  def rq_gripper_led_force_purple(gripper_socket="1"):
      rq_set_var(LBP,1, gripper_socket)
      rq_set_var(LRD,1, gripper_socket)
      rq_set_var(LBL,1, gripper_socket)
      rq_set_var(LGN,0, gripper_socket)
  end

  ############################################
  # mm/inches functions
  ############################################
  gripper_closed_norm = [100, 100, 100, 100]
  gripper_open_norm = [0, 0, 0, 0]
  gripper_closed_mm = [0, 0, 0, 0]
  gripper_open_mm = [50, 50, 50, 50]

  def rq_current_pos_mm(gripper_socket=1):
      pos_gripper = rq_current_pos(gripper_socket)
      pos_mm = gripper_to_mm(pos_gripper, gripper_socket)
      return round_value_2_dec(pos_mm)
  end

  def rq_current_pos_inches(gripper_socket=1):
      pos_gripper = rq_current_pos(gripper_socket)
      pos_mm = gripper_to_mm(pos_gripper, gripper_socket)
      pos_in = pos_mm / 25.4
      return round_value_2_dec(pos_in)
  end

  def rq_move_mm(pos_mm, gripper_socket=1):
      pos_gripper = mm_to_gripper(pos_mm, gripper_socket)
      rq_move(pos_gripper, gripper_socket)
  end

  def rq_move_and_wait_mm(pos_mm, gripper_socket=1):
      pos_gripper = mm_to_gripper(pos_mm, gripper_socket)
      rq_move_and_wait(pos_gripper, gripper_socket)
  end

  def rq_move_inches(pos_in, gripper_socket=1):
      pos_mm = pos_in * 25.4
      rq_move_mm(pos_mm, gripper_socket)
  end

  def rq_move_and_wait_inches(pos_in, gripper_socket=1):
      pos_mm = pos_in * 25.4
      rq_move_and_wait_mm(pos_mm, gripper_socket)
  end

  def get_closed_norm(gripper_socket):
      return gripper_closed_norm[gripper_socket - 1]
  end

  def get_open_norm(gripper_socket):
      return gripper_open_norm[gripper_socket - 1]
  end

  def get_closed_mm(gripper_socket):
      return gripper_closed_mm[gripper_socket - 1]
  end

  def get_open_mm(gripper_socket):
      return gripper_open_mm[gripper_socket - 1]
  end

  def set_closed_norm(closed_norm, gripper_socket):
      gripper_closed_norm[gripper_socket - 1] = closed_norm
  end

  def set_open_norm(open_norm, gripper_socket):
      gripper_open_norm[gripper_socket - 1] = open_norm
  end

  def set_closed_mm(closed_mm, gripper_socket):
      gripper_closed_mm[gripper_socket - 1] = closed_mm
  end

  def set_open_mm(open_mm, gripper_socket):
      gripper_open_mm[gripper_socket - 1] = open_mm
  end

  def gripper_to_mm(value_gripper, gripper_socket):
      closed_norm = get_closed_norm(gripper_socket)
      open_norm = get_open_norm(gripper_socket)
      closed_mm = get_closed_mm(gripper_socket)
      open_mm = get_open_mm(gripper_socket)

      value_norm = (value_gripper / 255) * 100

      slope = (closed_mm - open_mm) / (closed_norm - open_norm)
      value_mm = slope * (value_norm - closed_norm) + closed_mm

      if (value_mm > open_mm):
          value_mm_limited = open_mm
      elif (value_mm < closed_mm):
          value_mm_limited = closed_mm
      else:
          value_mm_limited = value_mm
      end

      return value_mm_limited
  end

  def mm_to_gripper(value_mm, gripper_socket):
      closed_norm = get_closed_norm(gripper_socket)
      open_norm = get_open_norm(gripper_socket)
      closed_mm = get_closed_mm(gripper_socket)
      open_mm = get_open_mm(gripper_socket)

      slope = (closed_norm - open_norm) / (closed_mm - open_mm)
      value_norm = (value_mm - closed_mm) * slope + closed_norm

      value_gripper = value_norm * 255 / 100

      if (value_gripper > 255):
          value_gripper_limited = 255
      elif (value_gripper < 0):
          value_gripper_limited = 0
      else:
          value_gripper_limited = round_value(value_gripper)
      end

      return value_gripper_limited
  end

  def round_value(value):
      value_mod = value % 1

      if(value_mod < 0.5):
          return floor(value)
      else:
          return ceil(value)
      end
  end

  def round_value_2_dec(value):
      value_x_100 = value * 100
      value_x_100_rounded = round_value(value_x_100)
      return value_x_100_rounded / 100
  end

  def clear_socket_buffer(gripper_socket="1", read_timeout = 0.1):
    byte_in_buffer = socket_read_byte_list(1, gripper_socket, read_timeout)

    while(byte_in_buffer[0] >= 1):
        byte_in_buffer = socket_read_byte_list(1, gripper_socket, read_timeout)
    end
  end

  def rq_set_gripper_socket_acquire_option(enabled=False):
      gripper_socket_acquire_option = enabled

      if(not enabled):
          gripper_1_socket_acquired = False
          gripper_2_socket_acquired = False
          gripper_3_socket_acquired = False
          gripper_4_socket_acquired = False
      end
  end

  def rq_acquire_gripper_socket(gripper_socket="1"):
      if(gripper_socket_acquire_option):
          rq_wait_gripper_socket_released(gripper_socket)
          enter_critical
              rq_set_gripper_socket_acquired(gripper_socket, True)
          exit_critical

          clear_socket_buffer(gripper_socket, 0.002)

          sync()
      end
  end

  def rq_release_gripper_socket(gripper_socket="1"):
      if(gripper_socket_acquire_option):
          rq_set_gripper_socket_acquired(gripper_socket, False)

          sync()
      end
  end

  def rq_set_gripper_socket_acquired(gripper_socket="1", acquired=False):
      if(gripper_socket == "1"):
          gripper_1_socket_acquired = acquired
      elif(gripper_socket == "2"):
          gripper_2_socket_acquired = acquired
      elif(gripper_socket == "3"):
          gripper_3_socket_acquired = acquired
      elif(gripper_socket == "4"):
          gripper_4_socket_acquired = acquired
      end
  end

  def rq_get_gripper_socket_acquired(gripper_socket="1"):
      if(gripper_socket == "1"):
          return gripper_1_socket_acquired
      elif(gripper_socket == "2"):
          return gripper_2_socket_acquired
      elif(gripper_socket == "3"):
          return gripper_3_socket_acquired
      elif(gripper_socket == "4"):
          return gripper_4_socket_acquired
      end

      sync()
  end

  def rq_wait_gripper_socket_released(gripper_socket="1"):
      while(rq_get_gripper_socket_acquired(gripper_socket)):
          sync()
      end

      sync()
  end

  def rq_gripper_id_to_ascii(gripper_id):
      if(gripper_id == "1"):
          return 57
      elif(gripper_id == "2"):
          return 50
      elif(gripper_id == "3"):
          return 51
      elif(gripper_id == "4"):
          return 52
      end
  end

  def scale(value, rawRange, scaledRange):
      def computeSlope(inputRange, outputRange):
          outputRangeDelta = outputRange[1] - outputRange[0]
          inputRangeDelta = inputRange[1] - inputRange[0]

          if (inputRangeDelta == 0):
              return 0
          else:
              return outputRangeDelta / inputRangeDelta
          end
      end

      def computeIntercept(slope, inputRange, outputRange):
          return outputRange[0] - (slope * inputRange[0])
      end

      def clipScaledValue(outputScaledValue, outputRange):
          if (outputRange[0] < outputRange[1]):
              return clipWhenLowerLimitIsLessThanHigher(outputScaledValue, outputRange)
          else:
              return clipWhenLowerLimitIsGreaterThanHigherLimit(outputScaledValue, outputRange)
          end
      end

      def clipWhenLowerLimitIsGreaterThanHigherLimit(outputScaledValue, outputRange):
          if (outputScaledValue < outputRange[1]):
              return outputRange[1]
          elif (outputScaledValue > outputRange[0]):
              return outputRange[0]
          else:
              return outputScaledValue
          end
      end

      def clipWhenLowerLimitIsLessThanHigher(outputScaledValue, outputRange):
          if (outputScaledValue < outputRange[0]):
              return outputRange[0]
          elif (outputScaledValue > outputRange[1]):
              return outputRange[1]
          else:
              return outputScaledValue
          end
      end

      slope = computeSlope(rawRange, scaledRange)
      intercept = computeIntercept(slope, rawRange, scaledRange)
      scaledValue = slope * value + intercept
      return clipScaledValue(scaledValue, scaledRange)
  end

  def limit(value, range):
      return scale(value, range, range)
  end


  rq_obj_detect = 0
  set_tool_voltage(24)
  set_tool_communication(True, 115200, 0, 1, 1.5, 3.5)
  rq_wait_for_gripper_connected()
  rq_init_comm_if_connected(9, "1")
  rq_init_comm_if_connected(2, "2")
  rq_init_comm_if_connected(3, "3")
  rq_init_comm_if_connected(4, "4")
  rq_print_connected_grippers()
  connectivity_checked = [-1,-1,-1,-1]
  status_checked = [-1,-1,-1,-1]
  current_speed = [-1,-1,-1,-1]
  current_force = [-1,-1,-1,-1]
  set_closed_norm(90.19607843137254, 1)
  set_open_norm(1.1764705882352942, 1)
  set_closed_mm(0.0, 1)
  set_open_mm(143.0, 1)
  set_closed_norm(100.0, 2)
  set_open_norm(0.0, 2)
  set_closed_mm(0.0, 2)
  set_open_mm(50.0, 2)
  set_closed_norm(100.0, 3)
  set_open_norm(0.0, 3)
  set_closed_mm(0.0, 3)
  set_open_mm(50.0, 3)
  set_closed_norm(100.0, 4)
  set_open_norm(0.0, 4)
  set_closed_mm(0.0, 4)
  set_open_mm(50.0, 4)
  # end: URCap Installation Node
  $ 1 "Robot Program"
  $ 2 "Script: artmDemofast_all.script"
      g_ftRaw = [0, 0, 0, 0, 0, 0, 0]
      g_transFlangeFts = pose_inv(p[0, 0, 0, 0, 0, 0])
      g_extFTRcv_stopReq = False
      g_filterOn = True

      set_payload(get_target_payload(), get_target_payload_cog())

      def filterData(a, b, currentPose, previousPose):
          counter = 0
          pose = currentPose
          if g_filterOn:
              while(counter < 6):
                  pose[counter] = (a * currentPose[counter] + b * previousPose[counter]) /(a + b)
                  counter = counter + 1
              end
          end
          return pose
      end

      thread extFTReceiverThread():
          prevData = p[0,0,0,0,0,0]
          while g_extFTRcv_stopReq == False:
              Error = 0
              ftRawData = get_tcp_force()
              ftRawData = filterData(0.002, 0.05, ftRawData, prevData)
              prevData = ftRawData

              flangePose = pose_inv(get_actual_tool_flange_pose())
              flangePose = p[0.0, 0.0, 0.0, flangePose[3], flangePose[4], flangePose[5]]

              ftDataForce = p[ftRawData[0], ftRawData[1], ftRawData[2], 0.0, 0.0, 0.0]
              ftDataForce = pose_trans(g_transFlangeFts,  pose_trans(flangePose, ftDataForce))

              ftDataTorque = p[ftRawData[3], ftRawData[4], ftRawData[5], 0.0, 0.0, 0.0]
              ftDataTorque = pose_trans(g_transFlangeFts, pose_trans(flangePose, ftDataTorque))
              enter_critical
              g_ftRaw = [Error, ftDataForce[0], ftDataForce[1], ftDataForce[2], ftDataTorque[0], ftDataTorque[1], ftDataTorque[2]]
              exit_critical
              sync()
          end
      end

      fts_rcv_thread = run extFTReceiverThread()

      # make sure we receive FT data
      while g_extFTRcv_stopReq == False:
          enter_critical
          tmpForceZ = g_ftRaw[3]
          exit_critical
          if tmpForceZ != 0:
             textmsg("ok, got some real force data")
             break
          end
          sync()
      end

      def killExtFTReceiverThread():
          kill fts_rcv_thread
      end
      g_ftRawBias_0 = 0
      g_ftRawBias_1 = 0
      g_ftRawBias_2 = 0
      g_ftRawBias_3 = 0
      g_ftRawBias_4 = 0
      g_ftRawBias_5 = 0
      def setExtFTBias():
          textmsg("Sleeping 0.1s to set Bias")
          sleep(0.1)
          # TODO: we need a more robust bias
          enter_critical
          local tmp = g_ftRaw
          exit_critical
          # use strongly smoothed data
          g_ftRawBias_0 = tmp[1]
          g_ftRawBias_1 = tmp[2]
          g_ftRawBias_2 = tmp[3]
          g_ftRawBias_3 = tmp[4]
          g_ftRawBias_4 = tmp[5]
          g_ftRawBias_5 = tmp[6]
          return tmp
      end

      def servojToTarget_132(target, a, v, t):
          local jp = get_target_joint_positions()
          i = 50
          if (t < 0.008):
              t = 0.008
          end
          while ((norm(jp[0] - target[0]) > 0.0006) or
                 (norm(jp[1] - target[1]) > 0.0006) or
                 (norm(jp[2] - target[2]) > 0.0006) or
                 (norm(jp[3] - target[3]) > 0.0006) or
                 (norm(jp[4] - target[4]) > 0.0006) or
                 (norm(jp[5] - target[5]) > 0.0006)) and (i > 0):
              if (evalGlobalConstraints_134()):
                  return True
              end
              servoj(target, a, v, t)
              jp = get_target_joint_positions()
              i = i - 1
          end
          if (i == 0):
              textmsg("servojToTarget: target not reached")
              halt
          end
      end

      def servojToTarget_123(target, a, v, t):
          local jp = get_target_joint_positions()
          i = 50
          if (t < 0.008):
              t = 0.008
          end
          while ((norm(jp[0] - target[0]) > 0.0006) or
                 (norm(jp[1] - target[1]) > 0.0006) or
                 (norm(jp[2] - target[2]) > 0.0006) or
                 (norm(jp[3] - target[3]) > 0.0006) or
                 (norm(jp[4] - target[4]) > 0.0006) or
                 (norm(jp[5] - target[5]) > 0.0006)) and (i > 0):
              if (evalGlobalConstraints_125()):
                  return True
              end
              servoj(target, a, v, t)
              jp = get_target_joint_positions()
              i = i - 1
          end
          if (i == 0):
              textmsg("servojToTarget: target not reached")
              halt
          end
      end


      socket_close("socket_gripper")
      socket_gripper_ok = socket_open("127.0.0.1", 63352, "socket_gripper")
      if socket_gripper_ok == False:
          # exit program/function
          halt
      end
      rps_rq_actual_pos = 1

      # Returns True if list_of_bytes is [3, 'a', 'c', 'k']
      def rps_is_ack(list_of_bytes):

          # list length is not 3
          if (list_of_bytes[0] != 3):
              return False
          end

          # first byte not is 'a'?
          if (list_of_bytes[1] != 97):
              return False
          end

          # first byte not is 'c'?
          if (list_of_bytes[2] != 99):
              return False
          end

          # first byte not is 'k'?
          if (list_of_bytes[3] != 107):
              return False
          end

          return True
      end

      def rps_rq_set_var(var_name, var_value):

          sync()
          socket_set_var(var_name , var_value, "socket_gripper")
          sync()
          ack = socket_read_byte_list(3, "socket_gripper")
          sync()

          while(not rps_is_ack(ack)):

              socket_set_var(var_name , var_value,"socket_gripper")
              sync()
              ack = socket_read_byte_list(3, "socket_gripper")
              sync()
          end
      end

      def rps_rq_get_var(var_name):

          if (var_name == "FLT"):
              socket_send_string("GET FLT","socket_gripper")
          elif (var_name == "OBJ"):
              socket_send_string("GET OBJ","socket_gripper")
          elif (var_name == "STA"):
              socket_send_string("GET STA","socket_gripper")
          elif (var_name == "PRE"):
              socket_send_string("GET PRE","socket_gripper")
          elif (var_name == "GTO"):
              socket_send_string("GET GTO", "socket_gripper")
          else:
              # nothing
          end

          sync()
          var_value = socket_read_byte_list(3, "socket_gripper")
          sync()

          return var_value
      end

      def rps_rq_set_GTO_sync(value):
          rps_rq_set_var("GTO",1)

          while (not rps_rq_is_GTO(value, rps_rq_get_var("GTO"))):
              sync()
          end
      end

      def rps_rq_is_GTO(value, bytes):
          asciiZero = 48

          if (bytes[0] == 1):
              if (bytes[1] == asciiZero + value):
                  return True
              end
          end

          return False
      end

      def regulateVacuum(maxLevel, timeout, minLevel):
          gripperPos = 0
          detectTimeout = 30
          advMode = False

          if (maxLevel == 0):
              gripperPos = 75
          elif (maxLevel == 1 and advMode):
              detectTimeout = 255
          end
          rps_rq_set_var("FOR", 100 - minLevel)
          rps_rq_set_var("POS", 100 - gripperPos)
          rps_rq_set_var("SPE", detectTimeout)

          rps_rq_set_var("MOD", 0)

          rps_rq_set_GTO_sync(1)
      end

      def rps_rq_get_position():

          rps_rq_actual_pos = 1
          if (rps_rq_is_object_detected()):
              rps_rq_actual_pos = 0
          end
          return rps_rq_actual_pos
      end

      # Returns True if list_of_byte is [1, '1'] or [1, '2']
      # Used to test OBJ = 0x1 or OBJ = 0x2
      def rps_is_OBJ_object_detected (list_of_bytes):
          # list length is not 1
          if (list_of_bytes[0] != 1):
              return False
          end

          # byte is '2'?
          if (list_of_bytes[1] == 50):
              return True
          end

          # byte is '1'?
          if (list_of_bytes[1] == 49):
              return True
          end

          return False
      end

      def rps_rq_wait_for_object_not_detected():
          while (rps_rq_is_object_detected()):
              sleep(0.01)
              sync()
          end
      end

      def rps_rq_wait_for_object_detected():
          while (not rps_rq_is_object_detected()):
              if (rps_rq_is_timeout()):
                  return False
              end
          end
          return True
      end

      def rps_rq_is_object_detected():
          gOBJ = rps_rq_get_var("OBJ")

          if(rps_is_OBJ_object_detected(gOBJ)):
              rps_rq_actual_pos = 0
              return True
          else:
              rps_rq_actual_pos = 1
              return False
          end
      end

      def rps_rq_is_timeout():
        return rps_rq_is_FLT(6, rps_rq_get_var("FLT"))
      end

      def rps_rq_is_FLT(fault_number, list_of_bytes):
          zero_ascii = 48
          if (list_of_bytes[0] != 2):
             return False
          end

          if (list_of_bytes[1] != zero_ascii):
              return False
          end

          if (list_of_bytes[2] != zero_ascii + fault_number):
              return False
          end

          return True
      end


      def rps_is_STA_gripper_activated(list_of_bytes):
          # list length is not 1
          if (list_of_bytes[0] != 1):
              return False
          end

          # byte is '3'?
          if (list_of_bytes[1] == 51):
              return True
          end
          return False
      end

      def rps_rq_is_gripper_activated():
          gSTA = rps_rq_get_var("STA")
          return rps_is_STA_gripper_activated(gSTA)
      end

      def rps_rq_activate():
          if (rps_rq_is_gripper_activated()):
              return True
          end
          popup("Gripper is not initialized. Initialize and continue?", title="Gripper Warning", warning=True, error=False, blocking=True)
          # reset
          rps_rq_mov_complete = 0
          rps_rq_obj_detect = 0
          rps_rq_actual_pos = 1
          rps_rq_set_var("ACT", 0)
          rps_rq_set_var("ATR", 0)
          sync()
          # activate
          rps_rq_set_var("ACT", 1)
          while (not rps_rq_is_gripper_activated()):
              # wait for activation completed
              sync()
          end
      end
      rps_rq_activate()
      rps_rq_get_position()

      def gripperMove(pos, speed, force):
          regulateVacuum(pos, speed, 65)

          if (pos == 1):
              global g_errorMoveGripper = False
          elif (pos == 0):
              global g_errorMoveGripper = not rps_rq_wait_for_object_detected()
          end

          return True
      end
      def gripperMoveV2(pos, speed):
          return gripperMove(pos, speed, 65)
      end


      global g_detector_pre_bytes = 4
      global g_detector_max_poses = 16    # determines the data size
      global g_detector_pose_bytes = 8
      global g_time_out_flag_vision = 0
      global g_detector_result = p[0,0,0,0,0,0]

      def RPS_socketTestVision(socket_ok, message):
          if socket_ok == 0:
              # exit program/function
              textmsg("The connection to the camera failed. The programm will be stopped.")
              #halt
              return 0
          else:
              textmsg(message)
              return 1
          end
      end

      def RPS_closeSocketsVision(socket_visor_ok, socket_visor_name):
          if socket_visor_ok == 1:
              socket_close(socket_visor_name)
              socket_visor_ok = 0
          end
          return socket_visor_ok
      end
      global g_detector_max_jobs_cognex = 99

      def sendToCognex(message1, message2, socket):
      	send_ok = socket_send_string(message1, socket)
      	send_ok = send_ok and socket_send_string(message2, socket)
      	send_ok = send_ok and socket_send_byte(13, socket)
      	send_ok = send_ok and socket_send_byte(10, socket)
      	return send_ok
      end

      def sendNumberToCognex(message1, number1, socket):
      	send_ok = socket_send_string(message1, socket)
      	send_ok = send_ok and socket_send_byte(48 + floor(number1 / 10), socket)
      	send_ok = send_ok and socket_send_byte(48 + (number1 % 10), socket)
      	send_ok = send_ok and socket_send_byte(13, socket)
      	send_ok = send_ok and socket_send_byte(10, socket)
      	return send_ok
      end

      def RPS_loginCognex(user, password, socket):
      	strWelcome = socket_read_line(socket)

      	strUser = socket_read_string(socket)
      	if sendToCognex(user, "", socket):
      		strPassword = socket_read_string(socket)
      		if sendToCognex(password, "", socket):
      			strUserLoggedIn = socket_read_line(socket)
      			if strUserLoggedIn == "User Logged In":
      				textmsg( strWelcome )
      				return 1
      			else:
      				textmsg("Login failed, user or password is invalid.")
      				return 0
      			end
      		end
      	end
      	textmsg("Login failed, couldn't send the login messages.")
      	return 0
      end

      def getAsciiToNumber_13_10(socket):
      #reads from a socket ASCII characters and generates Integers from it.
      #The numbers must end with the ASCII-bytes '13', '10'
      	i = 0
      	number = 0
      	sign = 1
      	while True:
      		ascii = socket_read_byte_list(1, socket)
      		if ascii[1] > 47 and ascii[1] < 58:
      			number = number * 10
      			number = number + (ascii[1] - 48)
      		elif ascii[1] == 240 and i == 0:
      			sign = -1
      		elif ascii[1] == 13:
      			ascii = socket_read_byte_list(1, socket)
      			if ascii[1] == 10:
      				return [1, number*sign]
      			else:
      				return [0, 0]
      			end
      		else:
      			return [0, 0]
      		end
      		i = i + 1
      	end
      	return [0, 0]
      end

      def setTriggerCognex(socket):
      	#holding time for the response of the trigger is 2s
      	if sendToCognex("SW8", "", socket):
      		strResponseSetTrg = socket_read_line(socket)
      		if strResponseSetTrg  == "1":
      			return 1
      		else:
      			textmsg("Trigger failed. The camera sent the following error code: ")
      			if strResponseSetTrg == "-2":
      				textmsg("-2: The command could not be executed.")
      				textmsg("Make sure that the trigger of the job is set to 'manual'.")
      			elif strResponseSetTrg == "-6":
      				textmsg("-6: User does not have 'Full Access' to execute the command.")
      			else:
      				textmsg(strResponseSetTrg)
      				textmsg("To decipher the code, please look into the cognex manual at Set Online in Basic Native Mode Communication")
      			end
      			return 0
      		end
      	else:
      		textmsg("Trigger failed, couldn't send the message.")
      		return 0
      	end
      end

      def setOnlineCognex(mode, socket):
      	if sendToCognex("SO", mode, socket):
      		strResponseSetOnl = socket_read_line(socket)
      		if strResponseSetOnl  == "1":
      			return 1
      		else:
      			textmsg("The camera online mode can't be set to: ", mode)
      			textmsg("Set Online failed. The camera sent the following error code: ")
      			if strResponseSetOnl == "-2":
      				textmsg("-2: The command could not be executed.")
      			elif strResponseSetOnl == "-5":
      				textmsg("-5: The communications flag was succesful but the sensor did not go Online because the sensor is set Offline manually.")
      				textmsg("The manual setting could be done through the In-Sight Explorer user interface or by a Discrete I/O signal.")
      			elif strResponseSetOnl == "-6":
      				textmsg("-6: User does not have 'Full Access' to execute the command.")
      			else:
      				textmsg(strResponseSetOnl)
      				textmsg("To decipher the code, please look into the cognex manual at Set Online in Basic Native Mode Communication")
      			end
      			return 0
      		end
      	else:
      		textmsg("Set Online failed, couldn't send the message.")
      		return 0
      	end
      end

      def getJobCognex(socket):
      	if sendToCognex("GJ", "", socket):
      		strResponseGetJob = socket_read_line(socket)
      		if strResponseGetJob  == "1":
      			numResponseGetJob = getAsciiToNumber_13_10(socket)
      			if numResponseGetJob[0] == 1: #actual Jobnumber == numResponseGetJob[1]
      				return numResponseGetJob
      			else:
      				textmsg("Get job failed, couldn't read the answer from the camera.")
      			end
      		else:
      			textmsg("Get job failed. The camera sent the following error code: ", strResponseGetJob)
      			textmsg("To decipher the code, please look into the cognex manual at Get Job in Basic Native Mode Communication")
      			return [0, 0]
      		end
      	else:
      		textmsg("Get job failed, couldn't send the message.")
      		return [0, 0]
      	end
      end

      def setJobCognex(jobnumber, socket):
      	if jobnumber > g_detector_max_jobs_cognex:
      		textmsg("The job index is higher than the supported number of jobs, which is ", g_detector_max_jobs_cognex)
      		return 0
      	end
      	setOnlineCognex("0", socket)
      	if sendNumberToCognex("SJ", jobnumber, socket): #consider timeout, if more than 2s load time
      		strSJ = ""
      		i = 0
      		while strSJ == "":
      			strSJ = socket_read_line(socket)
      			i = i + 1
      			if i == 3 and strSJ == "":
      				strSJ = "0"
      				textmsg("Job change failed. The camera didn't answer anymore.")
      			end
      		end
      		if strSJ == "1":
      			setOnlineCognex("1", socket)
      			return 1
      		else:
      			textmsg("Job change failed. Please check the job number.")
      			return 0
      		end
      	else:
      		textmsg("Job change failed, couldn't send the message.")
      		return 0
      	end
      end

      def invalidateCameraData():
      	sync()
      	# 4+g_detector_max_poses*8 entries
      	return [ 0,0,0,0, 0,0,0,0,0,0,0,0,  0,0,0,0,0,0,0,0,  0,0,0,0,0,0,0,0,  0,0,0,0,0,0,0,0,  0,0,0,0,0,0,0,0,  0,0,0,0,0,0,0,0,  0,0,0,0,0,0,0,0,  0,0,0,0,0,0,0,0,  0,0,0,0,0,0,0,0,  0,0,0,0,0,0,0,0,  0,0,0,0,0,0,0,0,  0,0,0,0,0,0,0,0,  0,0,0,0,0,0,0,0,  0,0,0,0,0,0,0,0,  0,0,0,0,0,0,0,0,  0,0,0,0,0,0,0,0]
      end

      def getOnlineCognex(socket):
      	if sendToCognex("GO", "", socket):
      		responseByteList = socket_read_line(socket)
      		if responseByteList  == "1":
      			return 1
      		elif responseByteList  == "0":
      			return 0
      		else:			#absorb possible other bugs
      			return 0
      		end
      	else:
      		textmsg("Get Online failed, couldn't send the message.")
      		return 0
      	end
      end

      def getNumberCognex(socket):
      	number = socket_read_ascii_float(1, socket, 20)
      	if number[0] == 0:
      		g_time_out_flag_vision = 1
      	end
      	return number[1]
      end


      def getCameraDataCognex(socket_visor_in, socket_visor_out):
      	local detector_data = [
      		0,0,0,0, 0,0,0,0,0,0,0,0,  0,0,0,0,0,0,0,0,  0,0,0,0,0,0,0,0,  0,0,0,0,0,0,0,0,  0,0,0,0,0,0,0,0,  0,0,0,0,0,0,0,0,  0,0,0,0,0,0,0,0,  0,0,0,0,0,0,0,0,  0,0,0,0,0,0,0,0,  0,0,0,0,0,0,0,0,  0,0,0,0,0,0,0,0,  0,0,0,0,0,0,0,0,  0,0,0,0,0,0,0,0,  0,0,0,0,0,0,0,0,  0,0,0,0,0,0,0,0,  0,0,0,0,0,0,0,0
      	] #the whole data of one job are saved in this data array.
      	detector_data[0] = 1  # the output is active
      	if setTriggerCognex(socket_visor_in):
      		detector_data[1] = 1  # triggered successful

      		g_time_out_flag_vision = 0

      		detector_data[2] = getNumberCognex(socket_visor_out) #number of active detectors / poses
      		if detector_data[2] == 0:
      			textmsg("The sum of enabled vision detectors is zero. Please activate at least one detector.")
      		end
      		if g_time_out_flag_vision == 1:
      			textmsg("A timeout error is detected. Go into the camera settings and increase the sleeptime for the jobchange.")
      			return detector_data
      		end

      		sumOfSuccesOfAllPoses = 0
      		i=0
      		while i < g_detector_max_poses:

      			detector_data[g_detector_pre_bytes + g_detector_pose_bytes*i + 0] = getNumberCognex(socket_visor_out) #communication-byte: detector is active
      			if detector_data[g_detector_pre_bytes + g_detector_pose_bytes*i + 0] == 1:

      				detector_data[g_detector_pre_bytes + g_detector_pose_bytes*i + 1] = getNumberCognex(socket_visor_out) #result of the detector, succes == 1 or fail == 0
      				if detector_data[g_detector_pre_bytes + g_detector_pose_bytes*i + 1] == 1:

      					sumOfSuccesOfAllPoses = sumOfSuccesOfAllPoses + 1
      					if sumOfSuccesOfAllPoses % 8 == 0:
      						sync()
      					end

      					detector_data[g_detector_pre_bytes + g_detector_pose_bytes*i + 2] = getNumberCognex(socket_visor_out)/1000	#Pos. X
      					detector_data[g_detector_pre_bytes + g_detector_pose_bytes*i + 3] = getNumberCognex(socket_visor_out)/1000	#Pos. Y
      					#detector_data[g_detector_pre_bytes + g_detector_pose_bytes*i + 4] = 0
      					#detector_data[g_detector_pre_bytes + g_detector_pose_bytes*i + 5] = 0
      					#detector_data[g_detector_pre_bytes + g_detector_pose_bytes*i + 6] = 0
      					detector_data[g_detector_pre_bytes + g_detector_pose_bytes*i + 7] = getNumberCognex(socket_visor_out)/180*3.14159 #(Yaw- )Angle in rad
      				end
      			end
      			if g_time_out_flag_vision == 1:
      				textmsg("A timeout error is detected. Please check the connection to the camera.")
      				textmsg("The transmission of the vision detector result with the following index failed: ", i)
      				if detector_data[g_detector_pre_bytes + g_detector_pose_bytes*i + 1] == 1:
      					detector_data[g_detector_pre_bytes + g_detector_pose_bytes*i + 1] = 0
      					sumOfSuccesOfAllPoses = sumOfSuccesOfAllPoses - 1
      				end
      				socket_read_string(socket_visor_out) #to read the remaining text out of the socket
      				return detector_data
      			end
      			i = i + 1
      		end
      		sync()
      		#if sumOfSuccesOfAllPoses == detector_data[2]:
      		#	detector_data[3] = 1
      		#else:
      		#	detector_data[3] = 0
      		#end
      		detector_data[3] = sumOfSuccesOfAllPoses
      		return detector_data
      	else:
      		textmsg("Sending Trigger to the Cognex camera failed. The program will be stopped.")
      		#detector_data[1] == 0 failed trigger
      		return detector_data
      	end
      end

      def getErrorMaxPose(index):
      	if index < g_detector_max_poses and index >= 0:
      		return True
      	elif index < 0:
      		textmsg("The index of the vision detector result is invalid. The minimal index is 0.")
      		return False
      	else:
      		textmsg("The index of the vision detector result is invalid. The maximal index is ", g_detector_max_poses-1)
      		return False
      	end
      end

      def getErrorPoseCognex(detectorByte, errorByte):
      	if detectorByte:
      		return errorByte
      	else:
      		textmsg("The index of the vision detector result is invalid. The detector isn't active.")
      		return 0
      	end
      end

      def boolToIntCognex(bool):
      	if bool == True:
      		return 1
      	else:
      		return 0
      	end
      end

      def changeJobRequestCognex(jobnumber, detector_job, ip_address_visor, socket_visor_in, socket_visor_out, socket_visor_out_ok, setJobSleepTime):
          #return-Value: [valid, detector_job, socket_visor_out_ok]
      	if getOnlineCognex(socket_visor_in) == 0:
      		if setOnlineCognex("1", socket_visor_in) == 0:
      			return [0, detector_job, socket_visor_out_ok]
      		end
      	end

      	if detector_job == jobnumber:
              # nothing changed
      		return [1, detector_job, socket_visor_out_ok]
      	else:
      		getJobResponse = getJobCognex(socket_visor_in)
      		if getJobResponse[0] == 1 and getJobResponse[1] == jobnumber: #Can only be true at the first program cycle of "changeJobRequestCognex" => the output socket must be open
      			socket_visor_out_ok = boolToIntCognex(socket_open(ip_address_visor, 3000, socket_visor_out))
      			if RPS_socketTestVision(socket_visor_out_ok, "successful connection: socket visor out") == 1:
      				return [1, jobnumber, socket_visor_out_ok]
      			else:
      				return [0, jobnumber, socket_visor_out_ok]
      			end
      		else:
      			if socket_visor_out_ok == 1:
      				socket_visor_out_ok = boolToIntCognex(RPS_closeSocketsVision(socket_visor_out_ok, socket_visor_out))
      			end
      			if setJobCognex(jobnumber, socket_visor_in):
      				#open the output socket, after this a short break, before the trigger command can follow
      				socket_visor_out_ok = boolToIntCognex(socket_open(ip_address_visor, 3000, socket_visor_out))
      				if RPS_socketTestVision(socket_visor_out_ok, "successful connection: socket visor out") == 1:
      					sleep(setJobSleepTime) #after Set Job (and before the trigger) a short break is necessary; cognex said it can need up to 2s
      					return [1, jobnumber, socket_visor_out_ok]
      				else:
      					return [0, jobnumber, socket_visor_out_ok]
      				end
      			else:
      				textmsg("Job can't be changed")
      				setOnlineCognex("1", socket_visor_in) #Set camera online otherwise it stays in state comms online? and rejects everything
      				return [0, detector_job, socket_visor_out_ok]
      			end
      		end
      	end
      end
      global g_detector_job_0 = -1
      global g_socket_visor_out_ok_0 =  0
      global g_socket_visor_in_ok_0 = boolToIntCognex(socket_open("192.168.0.1", 23, "socket_visor_in_0"))
      if RPS_socketTestVision(g_socket_visor_in_ok_0, "successfully connected to camera 0: socket visor in") == 0:
          halt
      end
      RPS_loginCognex("admin", "", "socket_visor_in_0")
      # 4+g_detector_max_poses*8 entries
      global g_detector_data_0_31 = [0,0,0,0,  0,0,0,0,0,0,0,0,  0,0,0,0,0,0,0,0,  0,0,0,0,0,0,0,0,  0,0,0,0,0,0,0,0,  0,0,0,0,0,0,0,0,  0,0,0,0,0,0,0,0,  0,0,0,0,0,0,0,0,  0,0,0,0,0,0,0,0,  0,0,0,0,0,0,0,0,  0,0,0,0,0,0,0,0,  0,0,0,0,0,0,0,0,  0,0,0,0,0,0,0,0,  0,0,0,0,0,0,0,0,  0,0,0,0,0,0,0,0,  0,0,0,0,0,0,0,0,  0,0,0,0,0,0,0,0]
      sync()

      def detectorRun_0_31(blocking):
          g_detector_data_0_31[3] = -1 # needed for detector_finished in detectorStatus
          returnValue = changeJobRequestCognex(31, g_detector_job_0, "192.168.0.1", "socket_visor_in_0", "socket_visor_out_0", g_socket_visor_out_ok_0, 0.5)
          valid = returnValue[0]
          g_detector_job_0 = returnValue[1]
          g_socket_visor_out_ok_0 = returnValue[2]
          if valid == 1:
              g_detector_data_0_31 = getCameraDataCognex("socket_visor_in_0", "socket_visor_out_0")
              valid = g_detector_data_0_31[1]  # Trigger-Value
          else:
              g_detector_data_0_31 = invalidateCameraData()
          end
          return valid == 1
      end


      def detectorGetResult_0_31(index):
      	g_detector_result = p[0, 0, 0, 0, 0, 0]
      	if getErrorMaxPose(index):
      		local indexBase = g_detector_pre_bytes + g_detector_pose_bytes * index
      		if getErrorPoseCognex(g_detector_data_0_31[indexBase+0], g_detector_data_0_31[indexBase+1]) == 1:
      			i = 2
      			while i < 8:
      				g_detector_result[i-2] = g_detector_data_0_31[indexBase+i]
      				i = i + 1
      				sync()
      			end
      			return True
      		end
      	end
      	return False
      end

      def moveManip_101():
          global g_errorMoveManip_101 = False
          movej([-0.539002, -1.97624, 2.154398, 4.5329461, -1.5680979, 1.032961], 3, 1)
          return True
      end
      sync()

      def pointModifier107():
          global g_point_mod_107 = genVar_104
          g_point_mod_107[0] = (g_point_mod_107[0] + 0.954)
          g_point_mod_107[1] = (g_point_mod_107[1] + -0.154)
          global genVar_108 = False
      end
      sync()

      def pointModifier109():
          global g_point_mod_109 = g_point_mod_107
          global genVar_110 = False
      end
      sync()

      def checkConstrCond111():
          global g_errorConstrCond_111 = False
          genVar_113 = frame_userVisionPoint
          global genVar_112 = True
          return True
          global genVar_112 = False
          global g_errorConstrCond_111 = not genVar_112
          return False
      end
      sync()

      g_pidJointPos_120 = get_actual_joint_positions()
      def moveCartesian_120(pose, time):
          global g_pidJointPos_120 = get_inverse_kin(pose_trans(pose_trans(p[-0, -0, -0, 0, 0, 0], frame_userPointBaseTrafo), pose))
          servoj(g_pidJointPos_120, 3, 0.75, time)
      end
      sync()

      def moveManip_120():
          global g_errorMoveManip_120 = False
          if (g_tcp != p[-8.9096233e-009, -7.5370039e-009, 0.125, -3.1415925, -5.6866583e-008, 1.0028153e-008]):
              global g_tcp = p[-8.9096233e-009, -7.5370039e-009, 0.125, -3.1415925, -5.6866583e-008, 1.0028153e-008]
              set_tcp(g_tcp)
              sync()
          end
          movel(pose_trans(pose_trans(p[-0, -0, -0, 0, 0, 0], frame_userPointBaseTrafo), p[1.595513e-006, 8.5946834e-007, -7.8893987e-007, -2.4052264e-007, -1.4088576e-007, 1.0509356e-006]), 1.2, 0.25)
          return True
      end
      sync()

      g_extForce_124 = p[0, 0, 0, 0, 0, 0]
      g_extTorque_124 = p[0, 0, 0, 0, 0, 0]
      g_ftsToTcpTransform_124 = p[0, 0, 0, 3.1415925, 5.6870832e-008, -1.0033215e-008]
      def getExtForceTorqueAsPose_124():
          enter_critical
          global g_ftRawSync = g_ftRaw
          exit_critical
          global g_extForce_124 = pose_trans(g_ftsToTcpTransform_124, p[(g_ftRawSync[1] - g_ftRawBias_0), (g_ftRawSync[2] - g_ftRawBias_1), (g_ftRawSync[3] - g_ftRawBias_2), 0, 0, 0])
      end
      sync()

      g_invStartPose_125 = p[0, 0, 0, 0, 0, 0]
      g_invStartOrientation_125 = p[0, 0, 0, 0, 0, 0]
      g_invPoseRef1_125 = p[-0, -0, -0, 0, 0, 0]
      g_ftExtents_125 = [1000, 1000, 50, 1000, 1000, 1000]
      g_forceRegTransform_125 = p[-0, -0, -75, 0, 0, 0]
      def evalGlobalConstraints_125():
          actualPose = get_actual_tcp_pose()
          getExtForceTorqueAsPose_124()
          global actualOrient = actualPose
          actualOrient[0] = 0
          actualOrient[1] = 0
          actualOrient[2] = 0
          e0_f = pose_trans(pose_trans(pose_trans(g_forceRegTransform_125, g_invStartOrientation_125), actualOrient), g_extForce_124)
          return (norm(e0_f[2]) <= g_ftExtents_125[2])
      end
      sync()

      g_startPose_123 = p[0, 0, 0, 0, 0, 0]
      g_pidJointPos_123 = get_actual_joint_positions()
      def moveCartesian_123(pose, time):
          global g_pidJointPos_123 = get_inverse_kin(pose_trans(g_startPose_123, pose))
          servoj(g_pidJointPos_123, 3, 0.75, time)
      end
      sync()

      def moveManip_123():
          global g_errorMoveManip_123 = False
          if (g_tcp != p[-8.9096233e-009, -7.5370039e-009, 0.125, -3.1415925, -5.6870832e-008, 1.0033215e-008]):
              global g_tcp = p[-8.9096233e-009, -7.5370039e-009, 0.125, -3.1415925, -5.6870832e-008, 1.0033215e-008]
              set_tcp(g_tcp)
              sync()
          end
          global g_invStartOrientation_125 = pose_inv(get_actual_tcp_pose())
          g_invStartOrientation_125[0] = 0
          g_invStartOrientation_125[1] = 0
          g_invStartOrientation_125[2] = 0
          global g_startPose_123 = get_actual_tcp_pose()
          loopCounter = 1
          while ((loopCounter <= 2273)):
              loopFraction = (loopCounter / 2273)
              moveCartesian_123(pose_trans(p[0, 0, 0, 0, 0, 0], interpolate_pose(p[3.1910295e-006, 1.7189282e-006, -1.5778837e-006, -4.8078186e-007, -2.8161401e-007, 2.1006845e-006], p[2.3471209e-006, 7.7436334e-007, -0.20000106, -3.902e-007, -9.2350668e-008, 5.7246262e-007], loopFraction)), 0.0020000001)
              if (evalGlobalConstraints_125()):
                  return True
              end
              loopCounter = (loopCounter + 1)
          end
          servojToTarget_123(g_pidJointPos_123, 3, 0.75, 0.0020000001)
          global g_errorMoveManip_123 = True
          return False
      end
      sync()

      g_startPose_127 = p[0, 0, 0, 0, 0, 0]
      g_pidJointPos_127 = get_actual_joint_positions()
      def moveCartesian_127(pose, time):
          global g_pidJointPos_127 = get_inverse_kin(pose_trans(g_startPose_127, pose))
          servoj(g_pidJointPos_127, 3, 0.75, time)
      end
      sync()

      def moveManip_127():
          global g_errorMoveManip_127 = False
          if (g_tcp != p[-8.9096233e-009, -7.5370039e-009, 0.125, -3.1415925, -5.6870821e-008, 1.0033205e-008]):
              global g_tcp = p[-8.9096233e-009, -7.5370039e-009, 0.125, -3.1415925, -5.6870821e-008, 1.0033205e-008]
              set_tcp(g_tcp)
              sync()
          end
          global g_startPose_127 = get_actual_tcp_pose()
          movel(pose_trans(g_startPose_127, p[1.5955152e-006, 8.5946238e-007, 0.19999921, -2.4034824e-007, -1.4078134e-007, 1.050144e-006]), 1.2, 0.25)
          return True
      end
      sync()

      def moveManip_129():
          global g_errorMoveManip_129 = False
          movej([0.12679601, -1.663906, 2.340214, 4.0346179, -1.569151, 1.699921], 3, 1)
          return True
      end
      sync()

      g_extForce_133 = p[0, 0, 0, 0, 0, 0]
      g_extTorque_133 = p[0, 0, 0, 0, 0, 0]
      g_ftsToTcpTransform_133 = p[0, 0, 0, 3.1415925, 5.6859601e-008, -1.0039416e-008]
      def getExtForceTorqueAsPose_133():
          enter_critical
          global g_ftRawSync = g_ftRaw
          exit_critical
          global g_extForce_133 = pose_trans(g_ftsToTcpTransform_133, p[(g_ftRawSync[1] - g_ftRawBias_0), (g_ftRawSync[2] - g_ftRawBias_1), (g_ftRawSync[3] - g_ftRawBias_2), 0, 0, 0])
      end
      sync()

      g_invStartPose_134 = p[0, 0, 0, 0, 0, 0]
      g_invStartOrientation_134 = p[0, 0, 0, 0, 0, 0]
      g_invPoseRef1_134 = p[-0, -0, -0, 0, 0, 0]
      g_ftExtents_134 = [1000, 1000, 50, 1000, 1000, 1000]
      g_forceRegTransform_134 = p[-0, -0, -55, 0, 0, 0]
      def evalGlobalConstraints_134():
          actualPose = get_actual_tcp_pose()
          getExtForceTorqueAsPose_133()
          global actualOrient = actualPose
          actualOrient[0] = 0
          actualOrient[1] = 0
          actualOrient[2] = 0
          e0_f = pose_trans(pose_trans(pose_trans(g_forceRegTransform_134, g_invStartOrientation_134), actualOrient), g_extForce_133)
          return (norm(e0_f[2]) <= g_ftExtents_134[2])
      end
      sync()

      g_startPose_132 = p[0, 0, 0, 0, 0, 0]
      g_pidJointPos_132 = get_actual_joint_positions()
      def moveCartesian_132(pose, time):
          global g_pidJointPos_132 = get_inverse_kin(pose_trans(g_startPose_132, pose))
          servoj(g_pidJointPos_132, 3, 0.75, time)
      end
      sync()

      def moveManip_132():
          global g_errorMoveManip_132 = False
          if (g_tcp != p[-8.9096233e-009, -7.5370039e-009, 0.125, -3.1415925, -5.6859601e-008, 1.0039416e-008]):
              global g_tcp = p[-8.9096233e-009, -7.5370039e-009, 0.125, -3.1415925, -5.6859601e-008, 1.0039416e-008]
              set_tcp(g_tcp)
              sync()
          end
          global g_invStartOrientation_134 = pose_inv(get_actual_tcp_pose())
          g_invStartOrientation_134[0] = 0
          g_invStartOrientation_134[1] = 0
          g_invStartOrientation_134[2] = 0
          global g_startPose_132 = get_actual_tcp_pose()
          loopCounter = 1
          while ((loopCounter <= 2273)):
              loopFraction = (loopCounter / 2273)
              moveCartesian_132(pose_trans(p[0, 0, 0, 0, 0, 0], interpolate_pose(p[1.2416232e-006, 2.5212203e-006, -5.4202934e-007, 4.8640197e-007, 8.4623019e-007, 2.3616087e-006], p[1.7607402e-006, 1.7317332e-006, -0.20000157, 3.7998742e-008, 1.4414347e-008, 2.0891487e-007], loopFraction)), 0.0020000001)
              if (evalGlobalConstraints_134()):
                  return True
              end
              loopCounter = (loopCounter + 1)
          end
          servojToTarget_132(g_pidJointPos_132, 3, 0.75, 0.0020000001)
          global g_errorMoveManip_132 = True
          return False
      end
      sync()

      g_startPose_136 = p[0, 0, 0, 0, 0, 0]
      g_pidJointPos_136 = get_actual_joint_positions()
      def moveCartesian_136(pose, time):
          global g_pidJointPos_136 = get_inverse_kin(pose_trans(g_startPose_136, pose))
          servoj(g_pidJointPos_136, 3, 0.75, time)
      end
      sync()

      def moveManip_136():
          global g_errorMoveManip_136 = False
          if (g_tcp != p[-8.9096233e-009, -7.5370039e-009, 0.125, -3.1415925, -5.6859058e-008, 1.0033888e-008]):
              global g_tcp = p[-8.9096233e-009, -7.5370039e-009, 0.125, -3.1415925, -5.6859058e-008, 1.0033888e-008]
              set_tcp(g_tcp)
              sync()
          end
          global g_startPose_136 = get_actual_tcp_pose()
          movel(pose_trans(g_startPose_136, p[6.2081978e-007, 1.2606104e-006, 0.19999973, 2.4326954e-007, 4.2323134e-007, 1.1811246e-006]), 1.2, 0.25)
          return True
      end
      sync()

      g_tcp = p[0, 0, 0, 0, 0, 0]
      set_tcp(g_tcp)
      sync()

      movej([-0.53902698, -1.976216, 2.154423, 4.5329809, -1.568074, 1.032937], 1, 0.1)
      gripperMoveV2(1, 0.2)
      genVar_100 = 0
      while ((genVar_100 <= 11)):
          if (moveManip_101()):
              textmsg("Constraints goal is valid (id 34)")
          else:
              textmsg("Constraints goal is invalid (id 34)")
          end
          genVar_103 = not detectorRun_0_31(True)
          if ((genVar_103 == False)):
              textmsg("Started job of detector")
          else:
              textmsg("Could not start job of detector")
              halt
          end
          genVar_105 = not detectorGetResult_0_31(0)
          genVar_104 = g_detector_result
          if ((genVar_105 == False)):
              textmsg("Retrieved result of job of detector")
          else:
              textmsg("Could not get result of job of detector")
          end
          genVar_106 = not genVar_105
          if (genVar_106):
              pointModifier107()
              pointModifier109()
              frame_userVisionPoint = g_point_mod_109
              if (checkConstrCond111()):
                  textmsg("Constraints goal is valid (id 111)")
              else:
                  textmsg("Constraints goal is invalid (id 111)")
              end
              if (not g_errorConstrCond_111):
                  frame_userVisionPoint = pose_trans(p[0, 0, 0, 0, 0, 0], frame_userVisionPoint)
                  genVar_115 = False
                  frame_userVisionPoint = pose_trans(frame_userVisionPoint, p[0, 0, 0, 0, 0, 0])
                  genVar_116 = False
                  frame_userVisionPoint = pose_trans(p[0, 0, 0, 0, 0, 0], frame_userVisionPoint)
                  genVar_117 = False
              end
          else:
              g_errorConstrCond_111 = False
          end
          genVar_118 = (genVar_105 or g_errorConstrCond_111)
          if (not genVar_118):
              frame_userPointBaseTrafo = pose_trans(frame_userVisionPoint, p[-0.95400274, 0.15401033, 0.13730308, -8.4232943e-006, -3.0173117e-006, 7.4426614e-005])
              genVar_119 = False
              if (moveManip_120()):
                  textmsg("Constraints goal is valid (id 47)")
              else:
                  textmsg("Constraints goal is invalid (id 47)")
              end
          end
          g_ftsBias_122 = setExtFTBias()
          if (moveManip_123()):
              textmsg("Constraints goal is valid (id 326)")
          else:
              textmsg("Constraints goal is invalid (id 326)")
              halt
          end
          g_errorMoveGripper_126 = False
          gripperMoveV2(0, 1)
          if (moveManip_127()):
              textmsg("Constraints goal is valid (id 451)")
          else:
              textmsg("Constraints goal is invalid (id 451)")
          end
          if (moveManip_129()):
              textmsg("Constraints goal is valid (id 473)")
          else:
              textmsg("Constraints goal is invalid (id 473)")
          end
          g_ftsBias_131 = setExtFTBias()
          if (moveManip_132()):
              textmsg("Constraints goal is valid (id 534)")
          else:
              textmsg("Constraints goal is invalid (id 534)")
              halt
          end
          g_errorMoveGripper_135 = False
          gripperMoveV2(1, 1)
          if (moveManip_136()):
              textmsg("Constraints goal is valid (id 621)")
          else:
              textmsg("Constraints goal is invalid (id 621)")
          end
          if (False):
              break
          end
          genVar_100 = (genVar_100 + 1)
      end
end
